// TIA Portal V20 export
DATA_BLOCK "J1_SCARA_Arm3D"   // DB11, Motion_DB
// stored: InstanceOfName TO_PositioningAxis, OfSystemLibElement TO_PositioningAxis, OfSystemLibVersion 9.0
TO_PositioningAxis   // technology object, version 9.0
   // // inherited from TO_SpeedAxis
   // // inherited from TO_Axis
   // // inherited from TO_Object
   // VAR
   //    Actor : TO_Struct_Actor;
   //    TorqueLimiting : TO_Struct_TorqueLimiting;
   //    LoadGear : TO_Struct_LoadGear;
   //    DynamicLimits : TO_Struct_DynamicLimits;
   //    DynamicDefaults : TO_Struct_DynamicDefaults;
   //    Override : TO_Struct_Override;
   //    ControlPanel : TO_Struct_ControlPanel;
   //    InternalToTrace : Array[1..4] of TO_Struct_Internal;
   //    Simulation : TO_Struct_AxisSimulation;
   // END_VAR
   // VAR
   //    Position { ExternalWritable := 'False'} : LReal;
   //    ActualPosition { ExternalWritable := 'False'} : LReal;
   //    ActualVelocity { ExternalWritable := 'False'} : LReal;
   //    ActualAcceleration { ExternalWritable := 'False'} : LReal;
   //    OperativeSensor { ExternalWritable := 'False'} : UDInt;
   //    ModuloCycle { ExternalWritable := 'False'} : DInt;
   //    ActualModuloCycle { ExternalWritable := 'False'} : DInt;
   //    Clamping { S7_SetPoint := 'True'} : TO_Struct_Clamping;
   //    Sensor { S7_SetPoint := 'True'} : Array[1..4] of TO_Struct_Sensor;
   //    Extrapolation { S7_SetPoint := 'True'} : TO_Struct_Extrapolation;
   //    Mechanics { S7_SetPoint := 'True'} : TO_Struct_Mechanics;
   //    Properties { ExternalWritable := 'False'; S7_SetPoint := 'True'} : TO_Struct_Properties;
   //    Modulo { S7_SetPoint := 'True'} : TO_Struct_Modulo;
   //    PositionLimits_SW { S7_SetPoint := 'True'} : TO_Struct_PositionLimitsSW;
   //    PositionLimits_HW { S7_SetPoint := 'True'} : TO_Struct_PositionLimitsHW;
   //    Homing { S7_SetPoint := 'True'} : TO_Struct_Homing;
   //    PositionControl { S7_SetPoint := 'True'} : TO_Struct_PositionControl;
   //    TorquePreControl { S7_SetPoint := 'True'} : TO_Struct_TorquePreControl;
   //    SetpointFilter { S7_SetPoint := 'True'} : TO_Struct_SetpointFilter;
   //    DynamicAxisModel { S7_SetPoint := 'True'} : TO_Struct_DynamicAxisModel;
   //    FollowingError { S7_SetPoint := 'True'} : TO_Struct_FollowingError;
   //    CrossPlcSynchronousOperation { S7_SetPoint := 'True'} : TO_Struct_CrossPlcSynchronousOperation;
   //    PositioningMonitoring { S7_SetPoint := 'True'} : TO_Struct_PositioningMonitoring;
   //    StandstillSignal { S7_SetPoint := 'True'} : TO_Struct_StandstillSignal;
   //    StatusPositioning { ExternalWritable := 'False'; S7_SetPoint := 'True'} : TO_Struct_StatusPositioning;
   //    StatusServo { ExternalWritable := 'False'; S7_SetPoint := 'True'} : TO_Struct_StatusServo;
   //    StatusProvidedLeadingValue { ExternalWritable := 'False'; S7_SetPoint := 'True'} : TO_Struct_StatusProvidedLeadingValue;
   //    StatusSensor { ExternalWritable := 'False'; S7_SetPoint := 'True'} : Array[1..4] of TO_Struct_StatusSensor;
   //    StatusExtrapolation { ExternalWritable := 'False'; S7_SetPoint := 'True'} : TO_Struct_StatusExtrapolation;
   //    StatusKinematicsMotion { ExternalWritable := 'False'; S7_SetPoint := 'True'} : TO_Struct_StatusKinematicsMotion;
   // END_VAR
BEGIN
   Actor.InverseDirection := false;
   Actor.Efficiency := 1.0;
   Actor.Interface.AddressIn.RID := 16#208072a;
   Actor.Interface.AddressOut.RID := 16#208072b;
   Actor.DriveParameter.ReferenceSpeed := 2000.0;
   Actor.DriveParameter.MaxSpeed := 2500.0;
   Actor.DriveParameter.ReferenceTorque := 23.9;
   TorqueLimiting.LimitBase := 1;
   TorqueLimiting.PositionBasedMonitorings := 0;
   TorqueLimiting.LimitDefaults.Torque := 0.0;
   TorqueLimiting.LimitDefaults.Force := 0.0;
   LoadGear.Numerator := 1348860;
   LoadGear.Denominator := 10000;
   DynamicLimits.MaxVelocity := 360.0;
   DynamicLimits.Velocity := 1000000000000.0;
   DynamicLimits.MaxAcceleration := 720.0;
   DynamicLimits.MaxDeceleration := 720.0;
   DynamicLimits.MaxJerk := 14400.0;
   DynamicDefaults.Velocity := 88.964;
   DynamicDefaults.Acceleration := 177.928;
   DynamicDefaults.Deceleration := 177.928;
   DynamicDefaults.Jerk := 24712.2222222222;
   DynamicDefaults.EmergencyDeceleration := 72000.0;
   Override.Velocity := 100.0;
   ControlPanel.Input.Command[1..2].ReqCounter := 0;
   ControlPanel.Input.Command[1..2]."Type" := 0;
   ControlPanel.Input.Command[1..2].Position := 0.0;
   ControlPanel.Input.Command[1..2].Velocity := 0.0;
   ControlPanel.Input.Command[1..2].Acceleration := 0.0;
   ControlPanel.Input.Command[1..2].Deceleration := 0.0;
   ControlPanel.Input.Command[1..2].Jerk := 0.0;
   ControlPanel.Input.Command[1..2].Param := 0.0;
   ControlPanel.Input.TimeOut := 2000.0;
   ControlPanel.Input.EsLifeSign := 0;
   InternalToTrace[1..4].Id := 0;
   InternalToTrace[1..4].Value := 0.0;
   Simulation.Mode := 1;
   Clamping.FollowingErrorDeviation := 360.0;
   Clamping.PositionTolerance := 360.0;
   Sensor[1]."Type" := 2;
   Sensor[1..4].InverseDirection := false;
   Sensor[1..4].System := 1;
   Sensor[1..4].MountingMode := 0;
   Sensor[2..4].DataAdaption := 0;
   Sensor[1].Interface.AddressIn.RID := 16#208072a;
   Sensor[1].Interface.AddressOut.RID := 16#208072b;
   Sensor[1..4].Parameter.Resolution := 0.001;
   Sensor[1].Parameter.StepsPerRevolution := 1024;
   Sensor[2..4].Parameter.StepsPerRevolution := 2048;
   Sensor[1..4].Parameter.FineResolutionXist1 := 11;
   Sensor[1].Parameter.FineResolutionXist2 := 0;
   Sensor[2..4].Parameter.FineResolutionXist2 := 9;
   Sensor[2..4].Parameter.DeterminableRevolutions := 1;
   Sensor[1..4].Parameter.DistancePerRevolution := 100.0;
   Sensor[1..4].Parameter.BehaviorGx_XIST1 := 0;
   Sensor[1..4].ActiveHoming.Mode := 0;
   Sensor[1..4].ActiveHoming.SideInput := true;
   Sensor[1..4].ActiveHoming.Direction := 0;
   Sensor[1..4].ActiveHoming.HomePositionOffset := 0.0;
   Sensor[1..4].ActiveHoming.SwitchLevel := true;
   Sensor[1..4].PassiveHoming.Mode := 0;
   Sensor[1..4].PassiveHoming.SideInput := true;
   Sensor[1..4].PassiveHoming.Direction := 2;
   Sensor[1..4].PassiveHoming.SwitchLevel := true;
   Extrapolation.FollowingAxisDependentTime := 0.0;
   Extrapolation.Settings.SystemDefinedExtrapolation := 1;
   Extrapolation.Settings.ExtrapolatedVelocityMode := 1;
   Extrapolation.PositionFilter.T1 := 0.0;
   Extrapolation.PositionFilter.T2 := 0.0;
   Extrapolation.VelocityFilter.T1 := 0.0;
   Extrapolation.VelocityFilter.T2 := 0.0;
   Extrapolation.VelocityTolerance.Range := 0.0;
   Extrapolation.Hysteresis.Value := 0.0;
   Mechanics.LeadScrew := 10.0;
   Properties.MotionType := 1;
   Modulo.Enable := false;
   Modulo.Length := 360.0;
   Modulo.StartValue := 0.0;
   PositionLimits_SW.Active := true;
   PositionLimits_SW.MinPosition := -160.0;
   PositionLimits_SW.MaxPosition := 160.0;
   PositionLimits_HW.Active := false;
   PositionLimits_HW.Mode := 1;
   PositionLimits_HW.MinSwitchLevel := true;
   PositionLimits_HW.MaxSwitchLevel := true;
   Homing.AutoReversal := false;
   Homing.ApproachDirection := false;
   Homing.ApproachVelocity := 3600.0;
   Homing.ReferencingVelocity := 900.0;
   Homing.HomePosition := 0.0;
   PositionControl.Kv := 100.0;
   PositionControl.Kpc := 100.0;
   PositionControl.EnableDSC := true;
   PositionControl.SmoothingTimeByChangeDifference := 0.0;
   PositionControl.InitialOperativeSensor := 1;
   PositionControl.ControlDifferenceQuantization.Mode := 1;
   PositionControl.ControlDifferenceQuantization.Value := 0.001;
   DynamicAxisModel.VelocityTimeConstant := 0.004;
   DynamicAxisModel.AdditionalPositionTimeConstant := 0.0;
   FollowingError.EnableMonitoring := true;
   FollowingError.MinValue := 360.0;
   FollowingError.MaxValue := 3600.0;
   FollowingError.MinVelocity := 360.0;
   FollowingError.WarningLevel := 70.0;
   CrossPlcSynchronousOperation.LocalLeadingValueDelayTime := 0.0;
   PositioningMonitoring.ToleranceTime := 1.0;
   PositioningMonitoring.MinDwellTime := 0.01;
   StandstillSignal.VelocityThreshold := 2.0;
   StandstillSignal.MinDwellTime := 0.01;
   _Properties.MotionType := 1;
   Sensor[1].Type := 2;
   _Actor.Interface.Telegram := 105;
   _Sensor[1].Interface.Telegram := 105;
END_DATA_BLOCK
